# EPICS substitutions: db/music_hv_FMF1.substitutions
#
# i.keshelashvili@gsi.de
#
file "db/music_hv.template"
{
    pattern { FC, CH }
            { 1,  0  }
            { 2,  1  }
}
